// Mitsubishi GX Works2 project: zone reset   PLC: FX1N/FX1NC

PROGRAM MAIN
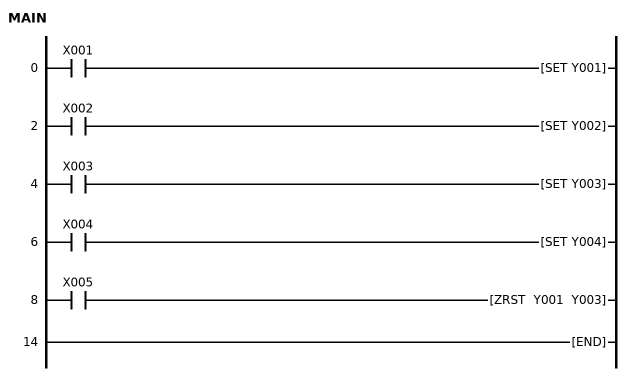
0     LD      X001
      SET     Y001
2     LD      X002
      SET     Y002
4     LD      X003
      SET     Y003
6     LD      X004
      SET     Y004
8     LD      X005
      ZRST    Y001 Y003
14    END
END_PROGRAM
